ABB RobotStudio station: w8.rspag

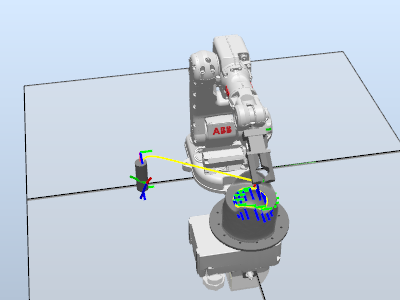
--- station ---
Station Project1 (saved by RobotStudio 22.3.10098.0)
Controller Controller1
  mechanical unit ROB_1: IRB140_6_81_C_03, 6 joints, base frame (0, 0, 0) mm
  mechanical unit M7DM1: MTD_250_M2009_REV1_01, 1 joints, base frame (584.98, -18.75, 250) mm, rotated rx 0 ry 0 rz 90 deg
Layout (positions relative to the parent item):
  - IRB140_6_81_C_03 [mechanism, from Robots\IRB140_6_81_C_G_03.rslib] at (0, 0, 0) mm; joint values [0, 0, 0, 0, 0.5236, 0] (rad or m)
  - MTD_250_M2009_REV1_01 [mechanism] at (584.98, -18.75, 250) mm, rotated rx 0 ry 0 rz 90 deg; joint values [0] (rad or m)
      links: Base, Link1
  - potty1 [part] at (698.66, 149.43, 241.77) mm, rotated rx 90 ry 0 rz 0 deg, size 275.1 x 194.8 x 257.3 mm
  - SmartComponent_1 [smart component, from Components\smart.rslib] at (506.29, 0, 679.5) mm, rotated rx 180 ry 60 rz 180 deg
      connections:
        SmartComponent_1.opengrip -> Detacher.Execute
        SmartComponent_1.closegrip -> Attacher.Execute
    - smart [mechanism, from Components\smart.rslib] at (0, 0, 0) mm
    - Attacher [smart component, from Components\Attacher.rslib]
        properties: Parent=smart; Flange=0; Child=tool-m2; Mount=false; Offset=[0 0 0]; Orientation=[0 0 0]
    - Detacher [smart component, from Components\Detacher.rslib]
        properties: Child=tool-m2; KeepPosition=false
  - tool-m2 [part] at (486.15, -642.32, 549.25) mm, size 50 x 50 x 143 mm
  - holder [part] at (486.15, -464.32, 428.25) mm, rotated rx 90 ry 0 rz 0 deg, size 50 x 120 x 49.5 mm
Attachment: potty1 is attached to MTD_250_M2009_REV1_01 / Link1
Attachment: potty is attached to potty1
Attachment: SmartComponent_1 is attached to IRB140_6_81_C_03 / Link6
Station logic (signal -> signal, property => property):
  Controller1.opengripper -> SmartComponent_1.opengrip
  Controller1.closegripper -> SmartComponent_1.closegrip

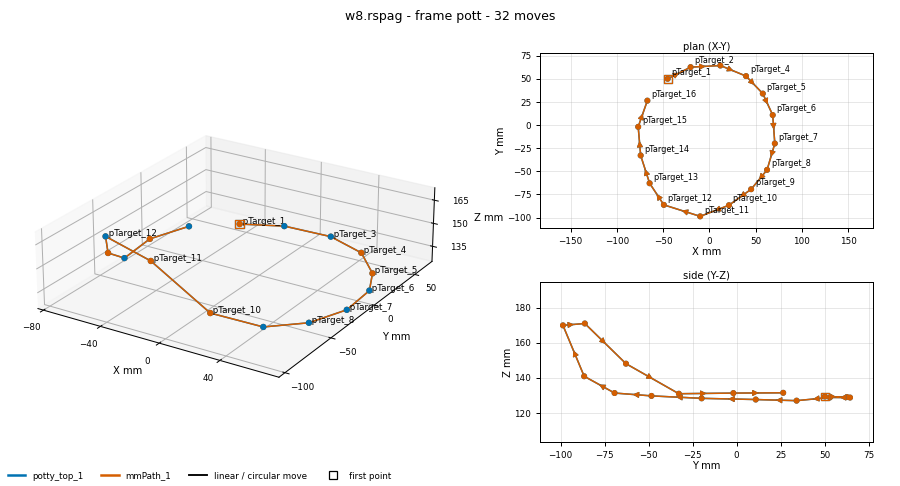
[picture p0: tool path of w8.rspag in frame pott, 32 of 42 moves have a stored position in this frame; points joined in program order, loops and branches not executed]
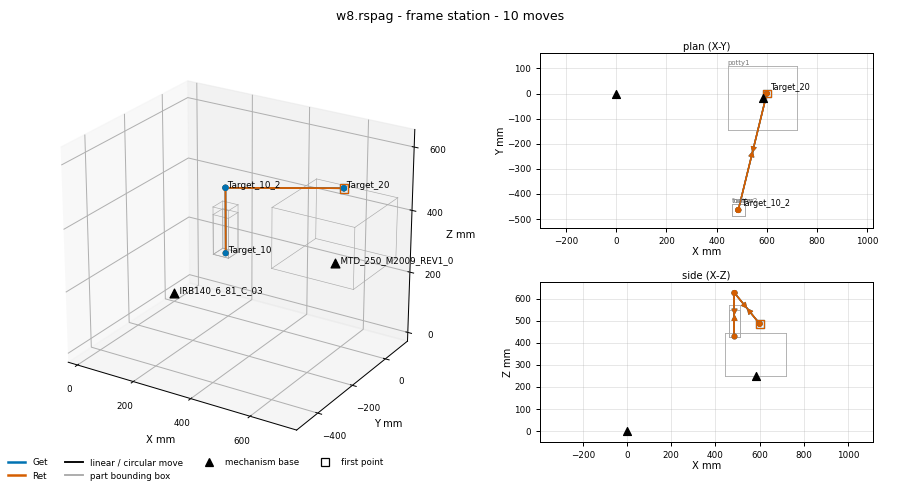
[picture p1: tool path of w8.rspag in frame station, 10 of 42 moves have a stored position in this frame; points joined in program order, loops and branches not executed]
--- Controller Data/Controller1/RAPID/TASK1/PROGMOD/CalibData.mod ---
MODULE CalibData
    PERS tooldata gripped_pen:=[TRUE,[[121,0,178],[1,0,0,0]],[2,[0,50,88],[1,0,0,0],0,0,0]];
    PERS wobjdata pott:=[FALSE,FALSE,"M7DM1",[[0,0,0],[1,0,0,0]],[[0,0,0],[1,0,0,0]]];
    TASK PERS wobjdata potty:=[FALSE,TRUE,"",[[584.978108354,-18.746939063,250],[0.707106781,0,0,0.707106781]],[[0,0,0],[1,0,0,0]]];
    PERS wobjdata w3_2:=[FALSE,FALSE,"M7DM1",[[0,0,0],[1,0,0,0]],[[0,0,0],[1,0,0,0]]];
    PERS tooldata smart:=[TRUE,[[121,0,178],[1,0,0,0]],[1.5,[0,77,66],[1,0,0,0],0,0,0]];
    TASK PERS wobjdata penholder:=[FALSE,TRUE,"ROB_1",[[516.431778047,-449.876609476,479.392371849],[0.26612336,0.822629428,-0.018923892,0.502096671]],[[0,0,0],[1,0,0,0]]];
ENDMODULE

--- Controller Data/Controller1/RAPID/TASK1/PROGMOD/Gripper.mod ---
MODULE Gripper(READONLY)
    PROC Opengrippers()
        Reset closegripper;
        Set opengripper;
    ENDPROC

    PROC Closegrippers()
        Reset opengripper;
        Set closegripper;
    ENDPROC
ENDMODULE

--- Controller Data/Controller1/RAPID/TASK1/PROGMOD/Module1.mod ---
MODULE Module1
        CONST robtarget pTarget_1:=[[-45.03,50.16,129.476],[0.5,0.5,0.5,-0.5],[-1,-1,0,1],[1.561940022,9E+09,9E+09,9E+09,9E+09,9E+09]];
    CONST robtarget pTarget_2:=[[-20.282,62.744,129.127],[0.5,0.5,0.5,-0.5],[-1,-1,0,1],[3.28998974,9E+09,9E+09,9E+09,9E+09,9E+09]];
    CONST robtarget pTarget_3:=[[11.896,64.483,128.86],[0.5,0.5,0.5,-0.5],[-1,-1,0,1],[5.728209081,9E+09,9E+09,9E+09,9E+09,9E+09]];
    CONST robtarget pTarget_4:=[[39.689,53.042,128.927],[0.5,0.5,0.5,-0.5],[-1,-1,0,1],[8.105863915,9E+09,9E+09,9E+09,9E+09,9E+09]];
    CONST robtarget pTarget_5:=[[57.798,34.115,127.1],[0.5,0.5,0.5,-0.5],[-1,-1,0,1],[10.023360048,9E+09,9E+09,9E+09,9E+09,9E+09]];
    CONST robtarget pTarget_6:=[[68.525,10.908,127.738],[0.5,0.5,0.5,-0.5],[-1,-1,0,1],[11.363158759,9E+09,9E+09,9E+09,9E+09,9E+09]];
    CONST robtarget pTarget_7:=[[70.794,-19.857,128.419],[0.5,0.5,0.5,-0.5],[0,-1,0,1],[12.181392468,9E+09,9E+09,9E+09,9E+09,9E+09]];
    CONST robtarget pTarget_8:=[[62.436,-48.353,129.808],[0.5,0.5,0.5,-0.5],[0,-1,0,1],[11.998377809,9E+09,9E+09,9E+09,9E+09,9E+09]];
    CONST robtarget pTarget_9:=[[45.201,-69.327,131.428],[0.5,0.5,0.5,-0.5],[-1,-1,0,1],[10.863368437,9E+09,9E+09,9E+09,9E+09,9E+09]];
    CONST robtarget pTarget_10:=[[21.201,-86.605,140.96],[0.5,0.5,0.5,-0.5],[-1,-1,0,1],[8.564003859,9E+09,9E+09,9E+09,9E+09,9E+09]];
    CONST robtarget pTarget_11:=[[-9.927,-98.657,169.887],[0.5,0.5,0.5,-0.5],[-1,-1,0,1],[4.189417321,9E+09,9E+09,9E+09,9E+09,9E+09]];
    CONST robtarget pTarget_12:=[[-49.23,-86.236,170.954],[0.5,0.5,0.5,-0.5],[-1,-1,0,1],[1.111919617,9E+09,9E+09,9E+09,9E+09,9E+09]];
    CONST robtarget pTarget_13:=[[-64.618,-62.853,148.116],[0.5,0.5,0.5,-0.5],[-1,-1,0,1],[1.685696862,9E+09,9E+09,9E+09,9E+09,9E+09]];
    CONST robtarget pTarget_14:=[[-74.299,-32.791,131.037],[0.5,0.5,0.5,-0.5],[-1,-1,0,1],[2.190066988,9E+09,9E+09,9E+09,9E+09,9E+09]];
    CONST robtarget pTarget_15:=[[-76.984,-1.82,131.395],[0.5,0.5,0.5,-0.5],[-1,-1,0,1],[2.117495861,9E+09,9E+09,9E+09,9E+09,9E+09]];
    CONST robtarget pTarget_16:=[[-67.051,26.501,131.572],[0.5,0.5,0.5,-0.5],[-1,-1,0,1],[2.848945135,9E+09,9E+09,9E+09,9E+09,9E+09]];
    CONST robtarget pTarget_17:=[[-45.03,50.16,129.476],[0.5,0.5,0.5,-0.5],[-1,-1,0,1],[4.22725007,9E+09,9E+09,9E+09,9E+09,9E+09]];
    CONST robtarget pTarget_18:=[[-20.282,62.744,129.127],[0.5,0.5,0.5,-0.5],[-1,-1,0,1],[6.076640279,9E+09,9E+09,9E+09,9E+09,9E+09]];
    CONST robtarget pTarget_19:=[[11.896,64.483,128.86],[0.5,0.5,0.5,-0.5],[-1,-1,0,1],[8.984552229,9E+09,9E+09,9E+09,9E+09,9E+09]];
    CONST robtarget pTarget_20:=[[39.689,53.042,128.927],[0.5,0.5,0.5,-0.5],[-1,-1,0,1],[12.005202323,9E+09,9E+09,9E+09,9E+09,9E+09]];
    CONST robtarget pTarget_21:=[[57.798,34.115,127.1],[0.5,0.5,0.5,-0.5],[-1,-1,0,1],[14.532593026,9E+09,9E+09,9E+09,9E+09,9E+09]];
    CONST robtarget pTarget_22:=[[68.525,10.908,127.738],[0.5,0.5,0.5,-0.5],[-1,-1,0,1],[16.42309869,9E+09,9E+09,9E+09,9E+09,9E+09]];
    CONST robtarget pTarget_23:=[[70.794,-19.857,128.419],[0.5,0.5,0.5,-0.5],[-1,-1,0,1],[17.790391273,9E+09,9E+09,9E+09,9E+09,9E+09]];
    CONST robtarget pTarget_24:=[[62.436,-48.353,129.808],[0.5,0.5,0.5,-0.5],[-1,-1,0,1],[17.994094103,9E+09,9E+09,9E+09,9E+09,9E+09]];
    CONST robtarget pTarget_25:=[[45.201,-69.327,131.428],[0.5,0.5,0.5,-0.5],[-1,-1,0,1],[17.05506634,9E+09,9E+09,9E+09,9E+09,9E+09]];
    CONST robtarget pTarget_26:=[[21.201,-86.605,140.96],[0.5,0.5,0.5,-0.5],[-1,-1,0,1],[14.920641693,9E+09,9E+09,9E+09,9E+09,9E+09]];
    CONST robtarget pTarget_27:=[[-9.927,-98.657,169.887],[0.5,0.5,0.5,-0.5],[-1,-1,0,1],[10.792580768,9E+09,9E+09,9E+09,9E+09,9E+09]];
    CONST robtarget pTarget_28:=[[-49.23,-86.236,170.954],[0.5,0.5,0.5,-0.5],[-1,-1,0,1],[7.02693357,9E+09,9E+09,9E+09,9E+09,9E+09]];
    CONST robtarget pTarget_29:=[[-64.618,-62.853,148.116],[0.5,0.5,0.5,-0.5],[-1,-1,0,1],[6.641524332,9E+09,9E+09,9E+09,9E+09,9E+09]];
    CONST robtarget pTarget_30:=[[-74.299,-32.791,131.037],[0.5,0.5,0.5,-0.5],[-1,-1,0,1],[6.185031074,9E+09,9E+09,9E+09,9E+09,9E+09]];
    CONST robtarget pTarget_31:=[[-76.984,-1.82,131.395],[0.5,0.5,0.5,-0.5],[-1,-1,0,1],[5.304441059,9E+09,9E+09,9E+09,9E+09,9E+09]];
    CONST robtarget pTarget_32:=[[-67.051,26.501,131.572],[0.5,0.5,0.5,-0.5],[-1,-1,0,1],[5.439420366,9E+09,9E+09,9E+09,9E+09,9E+09]];
    CONST robtarget Target_20:=[[152.846659375,-408.103868208,-139.614968698],[0.116673109,0.023513758,0.239931536,-0.963466318],[0,0,0,0],[0,9E+09,9E+09,9E+09,9E+09,9E+09]];
    CONST robtarget Target_10_2:=[[103.57736771,82.521620966,-69.777265452],[0.17479642,-0.226650886,0.201558845,-0.936722808],[-1,0,-1,0],[0,9E+09,9E+09,9E+09,9E+09,9E+09]];
    CONST robtarget Target_10:=[[-61.16522154,0.000000001,0.000000042],[0.17479642,-0.226650886,0.201558845,-0.936722808],[-1,1,-2,0],[0,9E+09,9E+09,9E+09,9E+09,9E+09]];
!***********************************************************
    !
    ! Module:  Module1
    !
    ! Description:
    !   <Insert description here>
    !
    ! Author: sgmxu9
    !
    ! Version: 1.0
    !
    !***********************************************************


    !***********************************************************
    !
    ! Procedure main
    !
    !   This is the entry point of your program
    !
    !***********************************************************
    PROC main()
        !Add your code here
        ActUnit M7DM1;
        Get;
        mmPath_1;
        Ret;
        DeactUnit M7DM1;
    ENDPROC
    PROC potty_top_1()
        ActUnit M7DM1;
        MoveL pTarget_1,v1000,z100,smart\WObj:=pott;
        MoveL pTarget_2,v1000,z100,smart\WObj:=pott;
        MoveL pTarget_3,v1000,z100,smart\WObj:=pott;
        MoveL pTarget_4,v1000,z100,smart\WObj:=pott;
        MoveL pTarget_5,v1000,z100,smart\WObj:=pott;
        MoveL pTarget_6,v1000,z100,smart\WObj:=pott;
        MoveL pTarget_7,v1000,z100,smart\WObj:=pott;
        MoveL pTarget_8,v1000,z100,smart\WObj:=pott;
        MoveL pTarget_9,v1000,z100,smart\WObj:=pott;
        MoveL pTarget_10,v1000,z100,smart\WObj:=pott;
        MoveL pTarget_11,v1000,z100,smart\WObj:=pott;
        MoveL pTarget_12,v1000,z100,smart\WObj:=pott;
        MoveL pTarget_13,v1000,z100,smart\WObj:=pott;
        MoveL pTarget_14,v1000,z100,smart\WObj:=pott;
        MoveL pTarget_15,v1000,z100,smart\WObj:=pott;
        MoveL pTarget_16,v1000,z100,smart\WObj:=pott;
    ENDPROC
    PROC mmPath_1()
        MoveJ pTarget_17,v1000,z100,smart\WObj:=pott;
        MoveL pTarget_18,v1000,z100,smart\WObj:=pott;
        MoveL pTarget_19,v1000,z100,smart\WObj:=pott;
        MoveL pTarget_20,v1000,z100,smart\WObj:=pott;
        MoveL pTarget_21,v1000,z100,smart\WObj:=pott;
        MoveL pTarget_22,v1000,z100,smart\WObj:=pott;
        MoveL pTarget_23,v1000,z100,smart\WObj:=pott;
        MoveL pTarget_24,v1000,z100,smart\WObj:=pott;
        MoveL pTarget_25,v1000,z100,smart\WObj:=pott;
        MoveL pTarget_26,v1000,z100,smart\WObj:=pott;
        MoveL pTarget_27,v1000,z100,smart\WObj:=pott;
        MoveL pTarget_28,v1000,z100,smart\WObj:=pott;
        MoveL pTarget_29,v1000,z100,smart\WObj:=pott;
        MoveL pTarget_30,v1000,z100,smart\WObj:=pott;
        MoveL pTarget_31,v1000,z100,smart\WObj:=pott;
        MoveL pTarget_32,v1000,z100,smart\WObj:=pott;
    ENDPROC
    PROC Get()
        MoveL Target_20,v1000,z100,smart\WObj:=penholder;
        MoveL Target_10_2,v1000,z100,smart\WObj:=penholder;
        MoveL Target_10,v1000,z100,smart\WObj:=penholder;
        WaitTime 1;
        Closegrippers;
        MoveL Target_10_2,v1000,z100,smart\WObj:=penholder;
        MoveL Target_20,v1000,z100,smart\WObj:=penholder;
    ENDPROC
    PROC Ret()
        MoveJ Target_20,v1000,z100,smart\WObj:=penholder;
        MoveL Target_10_2,v1000,z100,smart\WObj:=penholder;
        MoveL Target_10,v1000,z100,smart\WObj:=penholder;
        WaitTime 1;
        Opengrippers;
        MoveL Target_10_2,v1000,z100,smart\WObj:=penholder;
        MoveL Target_20,v1000,z100,smart\WObj:=penholder;
    ENDPROC
ENDMODULE

--- Controller Data/Controller1/SYSPAR/EIO.cfg ---
EIO:CFG_1.0:6:1::
#
INDUSTRIAL_NETWORK:

      -Name "DeviceNet" -Label "DeviceNet Master/Slave Network" -Address "2"
#
DEVICENET_DEVICE:

      -Name "board1" -VendorName "ABB Robotics" -ProductName "24 VDC I/O Device"\
      -Label "DSQC 652 24 VDC I/O Device" -ProductCode 26 -DeviceType 7\
      -ConnectionType "COS" -OutputSize 2 -InputSize 2
#
DEVICENET_INTERNAL_DEVICE:

      -Name "DN_Internal_Device" -VendorName "ABB Robotics"\
      -ProductName "DeviceNet Internal Slave Device"
#
EIO_SIGNAL:

      -Name "opengripper" -SignalType "DO" -Device "board1"\
      -Label "Open the Grippers" -DeviceMap "0" -Access "All"

      -Name "closegripper" -SignalType "DO" -Device "board1"\
      -Label "Close the Grippers" -DeviceMap "1" -Access "All"
